FUNCTION FC_RectFromSettings : TcVnRectangle_UDINT
VAR_INPUT
	setting:	ST_TEST_SETTING;
END_VAR
VAR
END_VAR

END_FUNCTION

(* stored: Version 1.1.0.1
   POU FC_RectFromSettings: Id {09c2f9b1-782c-44f8-9652-89340e25b543}, SpecialFunc None *)
